TYPE ST_HexMove_Input :
STRUCT
	t: LREAL;
END_STRUCT
END_TYPE

(* stored: Version 1.1.0.1, ProductVersion 3.1.4020.12
   DUT ST_HexMove_Input: Id {8f081c10-2d21-46ee-9ab4-59bfe335d0f0} *)
